{attribute 'GeneratedUsingTerminal: IODEVICETYPE_ETHERCATPROT'}
{attribute addProperty BoxType "IODEVICETYPE_ETHERCATPROT"}
{attribute addProperty Id "Beckhoff_EL1xxxBeckhoff_EL1xxx_E9115F816236Beckhoff_EL2xxxBeckhoff_EL2xxx_80BF8A152992Beckhoff_EL3xxxBeckhoff_EL3xxx_27F77F1B1813Beckhoff_EL3xxx_0030Beckhoff_EL3xxx_0030_1EE87FC6265Beckhoff_EL4xxxBeckhoff_EL4xxx_A204A3362405Beckhoff_EL5xxxBeckhoff_EL5xxx_51AF6A763086Beckhoff_EL6xxxBeckhoff_EL6xxx_C06944044115Beckhoff_EL7xxxBeckhoff_EL7xxx_2A642A8E2666Beckhoff_EL9xxxBeckhoff_EL9xxx_827611DB1254Beckhoff_EL15xxBeckhoff_EL15xx_B6DE29AF529Beckhoff_EL19xxBeckhoff_EL19xx_AAD37DB550Beckhoff_EL25xxBeckhoff_EL25xx_9005C0B32720Beckhoff_EL29xxBeckhoff_EL29xx_67A3BFC576Beckhoff_EL30xxBeckhoff_EL30xx_83B075E15129Beckhoff_EL31xxBeckhoff_EL31xx_33A6CB073694Beckhoff_EL32xxBeckhoff_EL32xx_54C941F72581Beckhoff_EL33xxBeckhoff_EL33xx_071A05C52459Beckhoff_EL34xxBeckhoff_EL34xx_534C4ABE11825Beckhoff_EL37xxBeckhoff_EL37xx_AD2113CE2253Beckhoff_EL47xxBeckhoff_EL47xx_E2BDD8A5294Beckhoff_EL66xxBeckhoff_EL66xx_168E4FCD1034Beckhoff_EL67xxBeckhoff_EL67xx_5C64E75D966Beckhoff_EL68xxBeckhoff_EL68xx_7666E5D03597Beckhoff_EL69xxBeckhoff_EL69xx_F00BD29B198Beckhoff_EL72xxBeckhoff_EL72xx_A73899913383Beckhoff_EL73xxBeckhoff_EL73xx_84A6DF1A1278Beckhoff_EL99xxBeckhoff_EL99xx_2141D83210SyncUnitsSyncUnits_9F8710E11242InputsInputs_25A0042B160OutputsOutputs_2397A10E106InfoDataInfoData_E68C61CD28"}
{attribute addProperty CRC "561887211"}
{attribute addProperty Size "68444"}
TYPE EtherCAT_Master_ELxxxx_217DB7EB :
STRUCT
	{attribute addProperty Name "Beckhoff_EL1xxx"}
	Beckhoff_EL1xxx : Beckhoff_EL1xxx_E9115F81;
	{attribute addProperty Name "Beckhoff_EL2xxx"}
	Beckhoff_EL2xxx : Beckhoff_EL2xxx_80BF8A15;
	{attribute addProperty Name "Beckhoff_EL3xxx"}
	Beckhoff_EL3xxx : Beckhoff_EL3xxx_27F77F1B;
	{attribute addProperty Name "Beckhoff_EL3xxx_0030"}
	Beckhoff_EL3xxx_0030 : Beckhoff_EL3xxx_0030_1EE87FC6;
	{attribute addProperty Name "Beckhoff_EL4xxx"}
	Beckhoff_EL4xxx : Beckhoff_EL4xxx_A204A336;
	{attribute addProperty Name "Beckhoff_EL5xxx"}
	Beckhoff_EL5xxx : Beckhoff_EL5xxx_51AF6A76;
	{attribute addProperty Name "Beckhoff_EL6xxx"}
	Beckhoff_EL6xxx : Beckhoff_EL6xxx_C0694404;
	{attribute addProperty Name "Beckhoff_EL7xxx"}
	Beckhoff_EL7xxx : Beckhoff_EL7xxx_2A642A8E;
	{attribute addProperty Name "Beckhoff_EL9xxx"}
	Beckhoff_EL9xxx : Beckhoff_EL9xxx_827611DB;
	{attribute addProperty Name "Beckhoff_EL15xx"}
	Beckhoff_EL15xx : Beckhoff_EL15xx_B6DE29AF;
	{attribute addProperty Name "Beckhoff_EL19xx"}
	Beckhoff_EL19xx : Beckhoff_EL19xx_AAD37DB5;
	{attribute addProperty Name "Beckhoff_EL25xx"}
	Beckhoff_EL25xx : Beckhoff_EL25xx_9005C0B3;
	{attribute addProperty Name "Beckhoff_EL29xx"}
	Beckhoff_EL29xx : Beckhoff_EL29xx_67A3BFC5;
	{attribute addProperty Name "Beckhoff_EL30xx"}
	Beckhoff_EL30xx : Beckhoff_EL30xx_83B075E1;
	{attribute addProperty Name "Beckhoff_EL31xx"}
	Beckhoff_EL31xx : Beckhoff_EL31xx_33A6CB07;
	{attribute addProperty Name "Beckhoff_EL32xx"}
	Beckhoff_EL32xx : Beckhoff_EL32xx_54C941F7;
	{attribute addProperty Name "Beckhoff_EL33xx"}
	Beckhoff_EL33xx : Beckhoff_EL33xx_071A05C5;
	{attribute addProperty Name "Beckhoff_EL34xx"}
	Beckhoff_EL34xx : Beckhoff_EL34xx_534C4ABE;
	{attribute addProperty Name "Beckhoff_EL37xx"}
	Beckhoff_EL37xx : Beckhoff_EL37xx_AD2113CE;
	{attribute addProperty Name "Beckhoff_EL47xx"}
	Beckhoff_EL47xx : Beckhoff_EL47xx_E2BDD8A5;
	{attribute addProperty Name "Beckhoff_EL66xx"}
	Beckhoff_EL66xx : Beckhoff_EL66xx_168E4FCD;
	{attribute addProperty Name "Beckhoff_EL67xx"}
	Beckhoff_EL67xx : Beckhoff_EL67xx_5C64E75D;
	{attribute addProperty Name "Beckhoff_EL68xx"}
	Beckhoff_EL68xx : Beckhoff_EL68xx_7666E5D0;
	{attribute addProperty Name "Beckhoff_EL69xx"}
	Beckhoff_EL69xx : Beckhoff_EL69xx_F00BD29B;
	{attribute addProperty Name "Beckhoff_EL72xx"}
	Beckhoff_EL72xx : Beckhoff_EL72xx_A7389991;
	{attribute addProperty Name "Beckhoff_EL73xx"}
	Beckhoff_EL73xx : Beckhoff_EL73xx_84A6DF1A;
	{attribute addProperty Name "Beckhoff_EL99xx"}
	Beckhoff_EL99xx : Beckhoff_EL99xx_2141D832;
	{attribute addProperty Name "SyncUnits"}
	SyncUnits : SyncUnits_9F8710E1;
	{attribute addProperty Name "Inputs"}
	Inputs : Inputs_25A0042B;
	{attribute addProperty Name "Outputs"}
	Outputs : Outputs_2397A10E;
	{attribute addProperty Name "InfoData"}
	InfoData : InfoData_E68C61CD;
END_STRUCT
END_TYPE

(* stored: Version 1.2.0.0, ProductVersion 3.1.4024.9
   DUT EtherCAT_Master_ELxxxx_217DB7EB: Id {c5e1903f-6ebb-468d-8c97-e2de864f6af4} *)
